(* PLC project LD_EVOLUTION_7, Beckhoff Automation GmbH TwinCAT PLC Control 3.5.10.30 *)
(* stored: creationDateTime 2019-09-26T16:32:19.6144365, modificationDateTime 2019-09-26T16:32:19.6144365 *)

PROGRAM Main
VAR
	A: BOOL;
	B: BOOL;
	Open: BOOL;
	C: BOOL;
	Count: BOOL;
END_VAR
  VAR  (* added by the conversion: wires and edge detectors of the diagram *)
    _EXECUTE7_EN : BOOL;
  END_VAR

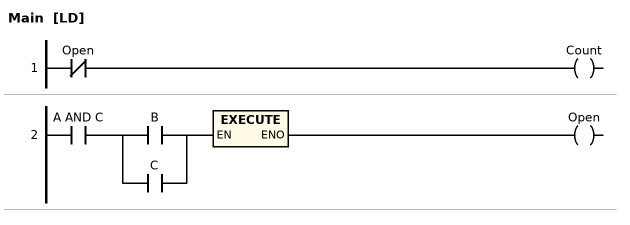
(* LD diagram, written out as Structured Text *)

Count := NOT Open;

_EXECUTE7_EN := (A AND C) AND (B OR C);
IF _EXECUTE7_EN THEN
  C:= A AND B;
  Open := C;
END_IF;
Open := _EXECUTE7_EN;
END_PROGRAM

CONFIGURATION Application
  RESOURCE LD_EVOLUTION_7 ON PLC
(* global variable list GVL *)
{attribute 'qualified_only'}
VAR_GLOBAL
	IsSFCResetting : BOOL;
END_VAR
    TASK PlcTask(INTERVAL := T#0ms, PRIORITY := 20);
    PROGRAM Main WITH PlcTask : Main;
  END_RESOURCE
END_CONFIGURATION
